// Mitsubishi GX Developer project: 电机顺序启停控制（二）   PLC: FX3U

PROGRAM MAIN
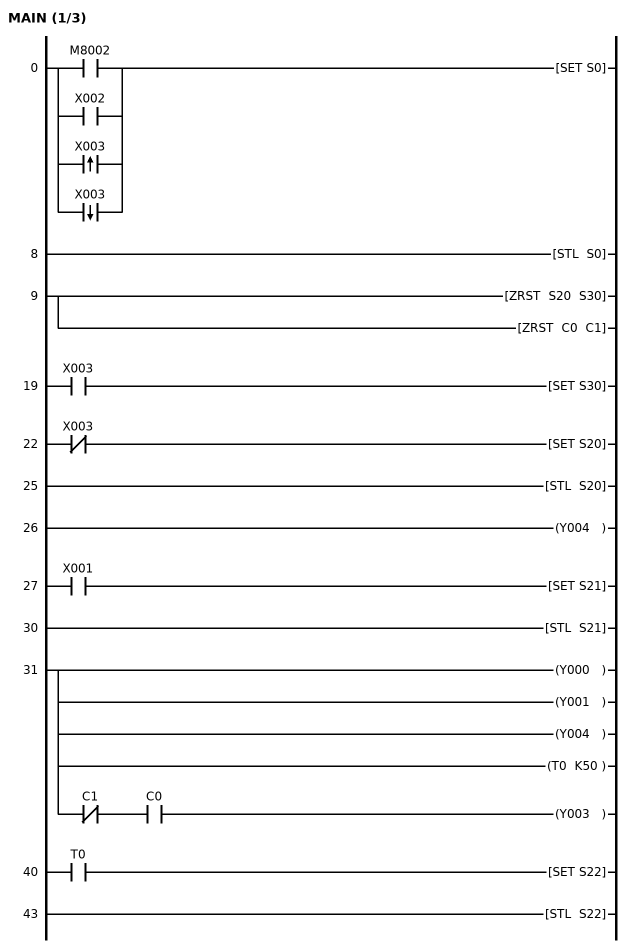
0     LD      M8002
      OR      X002
      ORP     X003
      ORF     X003
      SET     S0
8     STL     S0
9     ZRST    S20 S30
      ZRST    C0 C1
19    LD      X003
      SET     S30
22    LDI     X003
      SET     S20
25    STL     S20
26    OUT     Y004
27    LD      X001
      SET     S21
30    STL     S21
31    OUT     Y000
      OUT     Y001
      OUT     Y004
      OUT     T0 K50
      ANI     C1
      AND     C0
      OUT     Y003
40    LD      T0
      SET     S22
43    STL     S22
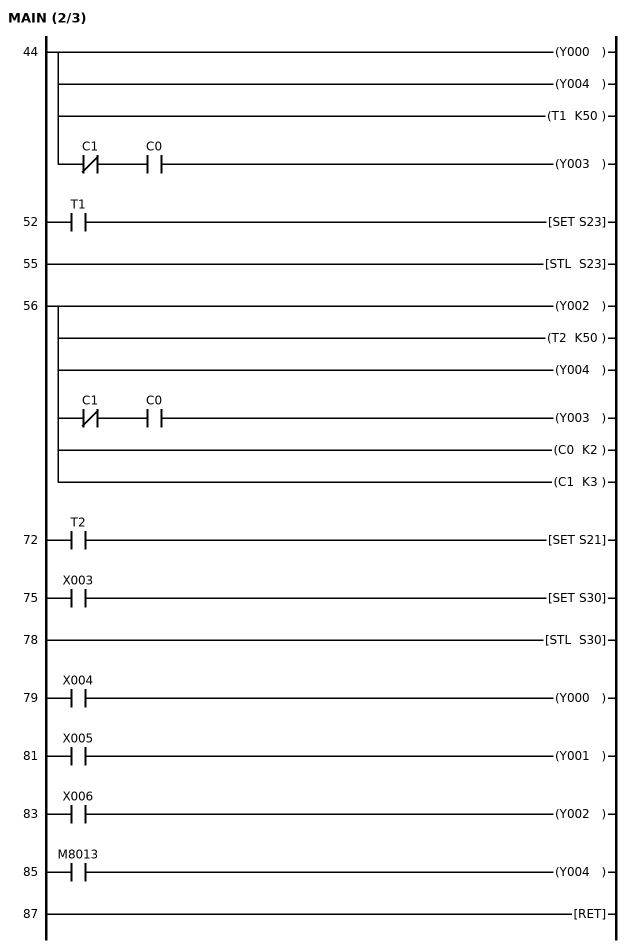
44    OUT     Y000
      OUT     Y004
      OUT     T1 K50
      ANI     C1
      AND     C0
      OUT     Y003
52    LD      T1
      SET     S23
55    STL     S23
56    OUT     Y002
      OUT     T2 K50
      OUT     Y004
      MPS
      ANI     C1
      AND     C0
      OUT     Y003
      MPP
      OUT     C0 K2
      OUT     C1 K3
72    LD      T2
      SET     S21
75    LD      X003
      SET     S30
78    STL     S30
79    LD      X004
      OUT     Y000
81    LD      X005
      OUT     Y001
83    LD      X006
      OUT     Y002
85    LD      M8013
      OUT     Y004
87    RET
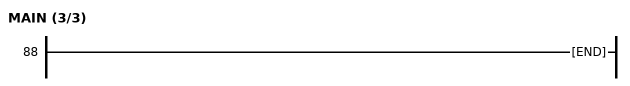
88    END
END_PROGRAM
